// TIA Portal project "Advanced Sorting by height (Working code)" (V17)

(* hardware
DEVICE "S71500/ET200MP-Station_1"  S7-1500 station
   slot 0: "Profilschiene_0"  6ES7 590-1***0-0AA0
   slot 1: "PLC_1"  CPU 1511-1 PN  6ES7 511-1AK00-0AB0  V1.8
   slot 2: "AI 8xU/I/RTD/TC ST_1"  AI 8xU/I/RTD/TC ST  6ES7 531-7KF00-0AB0  V2.0
   slot 3: "AI 8xU/I/RTD/TC ST_2"  AI 8xU/I/RTD/TC ST  6ES7 531-7KF00-0AB0  V2.0
   slot 4: "AI 8xU/I/RTD/TC ST_3"  AI 8xU/I/RTD/TC ST  6ES7 531-7KF00-0AB0  V2.0
   slot 5: "AI 8xU/I/RTD/TC ST_4"  AI 8xU/I/RTD/TC ST  6ES7 531-7KF00-0AB0  V2.0
   slot 6: "DI 16x24VDC BA_1"  DI 16x24VDC BA  6ES7 521-1BH10-0AA0  V1.0
*)

// ===== PLC "PLC_1"  CPU 1511-1 PN =====

VAR_GLOBAL   // PLC tag table "Standard-Variablentabelle"
   "At entry" AT %I0.0 : Bool;
   "Low box" AT %I0.1 : Bool;
   "High box" AT %I0.2 : Bool;
   "At turnable entry" AT %I0.3 : Bool;
   "At load position" AT %I0.4 : Bool;
   "At unload position" AT %I0.5 : Bool;
   "At front" AT %I0.6 : Bool;
   "At right entry" AT %I0.7 : Bool;
   "At left entry" AT %I1.0 : Bool;
   "At right exit" AT %I1.1 : Bool;
   "At left exit" AT %I1.2 : Bool;
   "Start" AT %I1.3 : Bool;
   "Reset" AT %I1.4 : Bool;
   "Stop" AT %I1.5 : Bool;
   "Emergency stop" AT %I1.6 : Bool;
   "Auto" AT %I1.7 : Bool;
   "Feeder Conveyor" AT %Q0.0 : Bool;
   "Entry Conveyor" AT %Q0.1 : Bool;
   "Load" AT %Q0.2 : Bool;
   "Unload" AT %Q0.3 : Bool;
   "Turn" AT %Q0.4 : Bool;
   "Left conveyor" AT %Q0.5 : Bool;
   "Right conveyor" AT %Q0.6 : Bool;
   "Green Indicator" AT %Q0.7 : Bool;
   "Yellow indicator" AT %Q1.0 : Bool;
   "Red indicator" AT %Q1.1 : Bool;
   "Start light" AT %Q1.2 : Bool;
   "Reset light" AT %Q1.3 : Bool;
   "Stop light" AT %Q1.4 : Bool;
   "Counter" AT %Q1.5 : Bool;
   "State 0" AT %M0.0 : Bool;
   "State 1" AT %M0.1 : Bool;
   "State 2" AT %M0.2 : Bool;
   "State 3" AT %M0.3 : Bool;
   "State 4" AT %M0.4 : Bool;
   "Factory IO Running" AT %I2.0 : Bool;
   "State 5" AT %M0.5 : Bool;
   "State 6" AT %M0.6 : Bool;
   "State 10" AT %M0.7 : Bool;
   "Low box detected" AT %M1.0 : Bool;
   "High box detected" AT %M1.1 : Bool;
   "Large box detected" AT %M1.2 : Bool;
   "Tag_1" AT %M2.0 : Bool;
   "Tag_2" AT %M2.1 : Bool;
   "Tag_3" AT %M2.2 : Bool;
   "Tag_6" AT %M2.3 : Bool;
   "Tag_9" AT %M2.4 : Bool;
   "Tag_10" AT %M2.5 : Bool;
   "Tag_11" AT %M2.6 : Bool;
   "Tag_12" AT %M2.7 : Bool;
   "Tag_14" AT %M3.0 : Bool;
   "Tag_15" AT %M3.1 : Bool;
   "Tag_16" AT %M3.2 : Bool;
   "Tag_17" AT %M3.3 : Bool;
   "Tag_18" AT %M3.4 : Bool;
   "Tag_19" AT %M4.0 : Bool;
   "Tag_20" AT %M5.0 : Bool;
END_VAR

FUNCTION "Start/Stop" : Void   // FC1, LAD
{ S7_Optimized_Access := 'TRUE' }
VERSION : 0.1
BEGIN

REGION Network 1: Start System
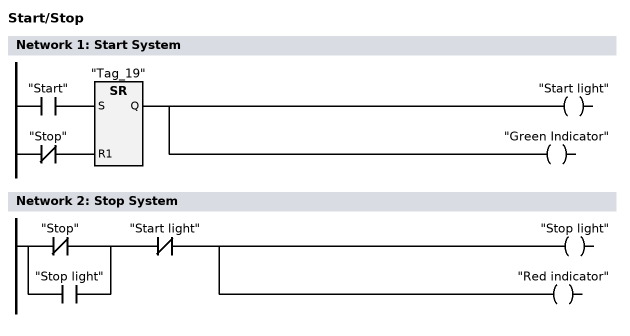
   RUNG wire#powerrail
      Contact( "Start" )
      S_SR(operand := "Tag_19", r1 := wire#w1)
      wire#w2
      Coil( "Start light" )
   END_RUNG
   RUNG wire#powerrail
      I_Contact( "Stop" )
   END_RUNG wire#w1
   RUNG wire#w2
      Coil( "Green Indicator" )
   END_RUNG
   // the same network as SCL:
   IF "Start" THEN
       "Tag_19" := TRUE;   // SR flip-flop
   END_IF;
   IF NOT "Stop" THEN "Tag_19" := FALSE; END_IF;
   "Start light" := "Tag_19";
   "Green Indicator" := "Tag_19";
END_REGION

REGION Network 2: Stop System
   RUNG wire#powerrail
      I_Contact( "Stop" )
      wire#w1
      I_Contact( "Start light" )
      wire#w2
      Coil( "Stop light" )
   END_RUNG
   RUNG wire#powerrail
      Contact( "Stop light" )
   END_RUNG wire#w1
   RUNG wire#w2
      Coil( "Red indicator" )
   END_RUNG
   // the same network as SCL:
   "Stop light" := (NOT "Stop" OR "Stop light") AND NOT "Start light";
   "Red indicator" := "Stop light";
END_REGION
END_FUNCTION

FUNCTION "States" : Void   // FC2, LAD
TITLE = States of the
{ S7_Optimized_Access := 'TRUE' }
VERSION : 0.1
// In this Programm, we will make every actuator is a state, and we will focus on Set Reset conditions, 
// POV : we will not consider which first and which after because it isn't recurrent
   VAR_TEMP   // added for the SCL form of the ladder/FBD networks
      _w1 : Bool;
      _w2 : Bool;
   END_VAR
BEGIN

REGION Network 1: Reset Loop
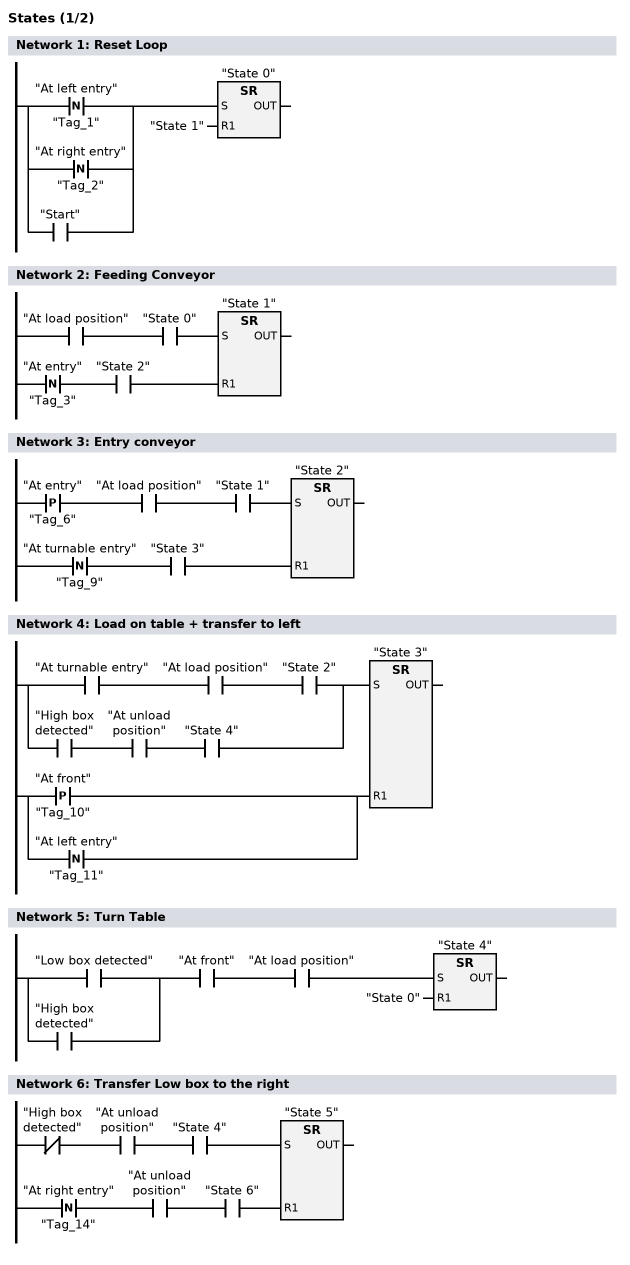
   RUNG wire#powerrail
      N_Contact(operand := "At left entry", bit := "Tag_1")
      wire#w1
      S_SR(operand := "State 0", r1 := "State 1")
   END_RUNG
   RUNG wire#powerrail
      N_Contact(operand := "At right entry", bit := "Tag_2")
   END_RUNG wire#w1
   RUNG wire#powerrail
      Contact( "Start" )
   END_RUNG wire#w1
   // the same network as SCL:
   #_w1 := NOT "At left entry" AND "Tag_1";   // falling edge of "At left entry"
   "Tag_1" := "At left entry";
   #_w2 := NOT "At right entry" AND "Tag_2";   // falling edge of "At right entry"
   "Tag_2" := "At right entry";
   IF #_w1 OR #_w2 OR "Start" THEN
       "State 0" := TRUE;   // SR flip-flop
   END_IF;
   IF "State 1" THEN "State 0" := FALSE; END_IF;
END_REGION

REGION Network 2: Feeding Conveyor
   RUNG wire#powerrail
      Contact( "At load position" )
      Contact( "State 0" )
      S_SR(operand := "State 1", r1 := wire#w1)
   END_RUNG
   RUNG wire#powerrail
      N_Contact(operand := "At entry", bit := "Tag_3")
      Contact( "State 2" )
   END_RUNG wire#w1
   // the same network as SCL:
   #_w1 := NOT "At entry" AND "Tag_3";   // falling edge of "At entry"
   "Tag_3" := "At entry";
   IF "At load position" AND "State 0" THEN
       "State 1" := TRUE;   // SR flip-flop
   END_IF;
   IF #_w1 AND "State 2" THEN "State 1" := FALSE; END_IF;
END_REGION

REGION Network 3: Entry conveyor
   RUNG wire#powerrail
      P_Contact(operand := "At entry", bit := "Tag_6")
      Contact( "At load position" )
      Contact( "State 1" )
      S_SR(operand := "State 2", r1 := wire#w1)
   END_RUNG
   RUNG wire#powerrail
      N_Contact(operand := "At turnable entry", bit := "Tag_9")
      Contact( "State 3" )
   END_RUNG wire#w1
   // the same network as SCL:
   #_w1 := "At entry" AND NOT "Tag_6";   // rising edge of "At entry"
   "Tag_6" := "At entry";
   #_w2 := NOT "At turnable entry" AND "Tag_9";   // falling edge of "At turnable entry"
   "Tag_9" := "At turnable entry";
   IF #_w1 AND "At load position" AND "State 1" THEN
       "State 2" := TRUE;   // SR flip-flop
   END_IF;
   IF #_w2 AND "State 3" THEN "State 2" := FALSE; END_IF;
END_REGION

REGION Network 4: Load on table + transfer to left
   RUNG wire#powerrail
      Contact( "At turnable entry" )
      Contact( "At load position" )
      Contact( "State 2" )
      wire#w1
      S_SR(operand := "State 3", r1 := wire#w2)
   END_RUNG
   RUNG wire#powerrail
      Contact( "High box detected" )
      Contact( "At unload position" )
      Contact( "State 4" )
   END_RUNG wire#w1
   RUNG wire#powerrail
      P_Contact(operand := "At front", bit := "Tag_10")
   END_RUNG wire#w2
   RUNG wire#powerrail
      N_Contact(operand := "At left entry", bit := "Tag_11")
   END_RUNG wire#w2
   // the same network as SCL:
   #_w1 := "At front" AND NOT "Tag_10";   // rising edge of "At front"
   "Tag_10" := "At front";
   #_w2 := NOT "At left entry" AND "Tag_11";   // falling edge of "At left entry"
   "Tag_11" := "At left entry";
   IF ("At turnable entry" AND "At load position" AND "State 2") OR ("High box detected" AND "At unload position" AND "State 4") THEN
       "State 3" := TRUE;   // SR flip-flop
   END_IF;
   IF #_w1 OR #_w2 THEN "State 3" := FALSE; END_IF;
END_REGION

REGION Network 5: Turn Table
   RUNG wire#powerrail
      Contact( "Low box detected" )
      wire#w1
      Contact( "At front" )
      Contact( "At load position" )
      S_SR(operand := "State 4", r1 := "State 0")
   END_RUNG
   RUNG wire#powerrail
      Contact( "High box detected" )
   END_RUNG wire#w1
   // the same network as SCL:
   IF ("Low box detected" OR "High box detected") AND "At front" AND "At load position" THEN
       "State 4" := TRUE;   // SR flip-flop
   END_IF;
   IF "State 0" THEN "State 4" := FALSE; END_IF;
END_REGION

REGION Network 6: Transfer Low box to the right
   RUNG wire#powerrail
      I_Contact( "High box detected" )
      Contact( "At unload position" )
      Contact( "State 4" )
      S_SR(operand := "State 5", r1 := wire#w1)
   END_RUNG
   RUNG wire#powerrail
      N_Contact(operand := "At right entry", bit := "Tag_14")
      Contact( "At unload position" )
      Contact( "State 6" )
   END_RUNG wire#w1
   // the same network as SCL:
   #_w1 := NOT "At right entry" AND "Tag_14";   // falling edge of "At right entry"
   "Tag_14" := "At right entry";
   IF NOT "High box detected" AND "At unload position" AND "State 4" THEN
       "State 5" := TRUE;   // SR flip-flop
   END_IF;
   IF #_w1 AND "At unload position" AND "State 6" THEN "State 5" := FALSE; END_IF;
END_REGION

REGION Network 7: Right conveyor
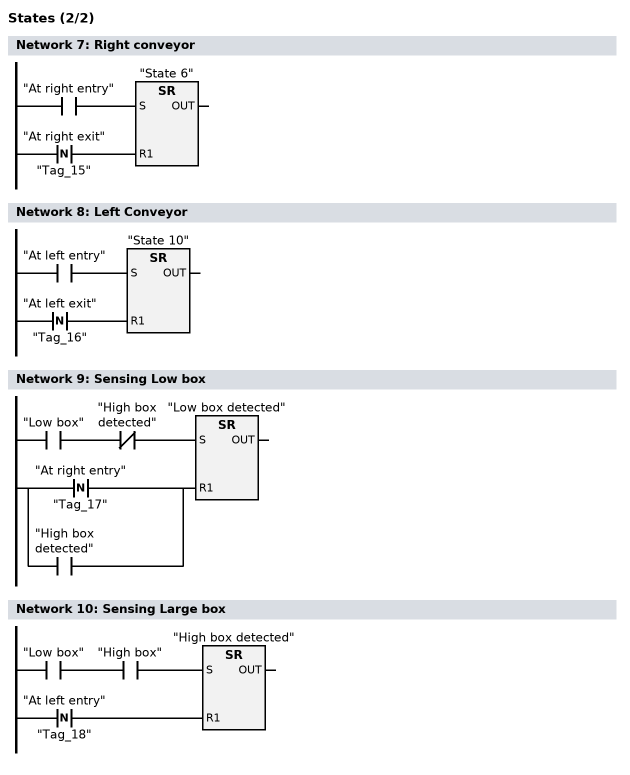
   RUNG wire#powerrail
      Contact( "At right entry" )
      S_SR(operand := "State 6", r1 := wire#w1)
   END_RUNG
   RUNG wire#powerrail
      N_Contact(operand := "At right exit", bit := "Tag_15")
   END_RUNG wire#w1
   // the same network as SCL:
   #_w1 := NOT "At right exit" AND "Tag_15";   // falling edge of "At right exit"
   "Tag_15" := "At right exit";
   IF "At right entry" THEN
       "State 6" := TRUE;   // SR flip-flop
   END_IF;
   IF #_w1 THEN "State 6" := FALSE; END_IF;
END_REGION

REGION Network 8: Left Conveyor
   RUNG wire#powerrail
      Contact( "At left entry" )
      S_SR(operand := "State 10", r1 := wire#w1)
   END_RUNG
   RUNG wire#powerrail
      N_Contact(operand := "At left exit", bit := "Tag_16")
   END_RUNG wire#w1
   // the same network as SCL:
   #_w1 := NOT "At left exit" AND "Tag_16";   // falling edge of "At left exit"
   "Tag_16" := "At left exit";
   IF "At left entry" THEN
       "State 10" := TRUE;   // SR flip-flop
   END_IF;
   IF #_w1 THEN "State 10" := FALSE; END_IF;
END_REGION

REGION Network 9: Sensing Low box
   RUNG wire#powerrail
      Contact( "Low box" )
      I_Contact( "High box detected" )
      S_SR(operand := "Low box detected", r1 := wire#w1)
   END_RUNG
   RUNG wire#powerrail
      N_Contact(operand := "At right entry", bit := "Tag_17")
   END_RUNG wire#w1
   RUNG wire#powerrail
      Contact( "High box detected" )
   END_RUNG wire#w1
   // the same network as SCL:
   #_w1 := NOT "At right entry" AND "Tag_17";   // falling edge of "At right entry"
   "Tag_17" := "At right entry";
   IF "Low box" AND NOT "High box detected" THEN
       "Low box detected" := TRUE;   // SR flip-flop
   END_IF;
   IF #_w1 OR "High box detected" THEN "Low box detected" := FALSE; END_IF;
END_REGION

REGION Network 10: Sensing Large box
   RUNG wire#powerrail
      Contact( "Low box" )
      Contact( "High box" )
      S_SR(operand := "High box detected", r1 := wire#w1)
   END_RUNG
   RUNG wire#powerrail
      N_Contact(operand := "At left entry", bit := "Tag_18")
   END_RUNG wire#w1
   // the same network as SCL:
   #_w1 := NOT "At left entry" AND "Tag_18";   // falling edge of "At left entry"
   "Tag_18" := "At left entry";
   IF "Low box" AND "High box" THEN
       "High box detected" := TRUE;   // SR flip-flop
   END_IF;
   IF #_w1 THEN "High box detected" := FALSE; END_IF;
END_REGION
END_FUNCTION

FUNCTION "Actuators" : Void   // FC3, LAD
{ S7_Optimized_Access := 'TRUE' }
VERSION : 0.1
BEGIN

REGION Network 1: State 0
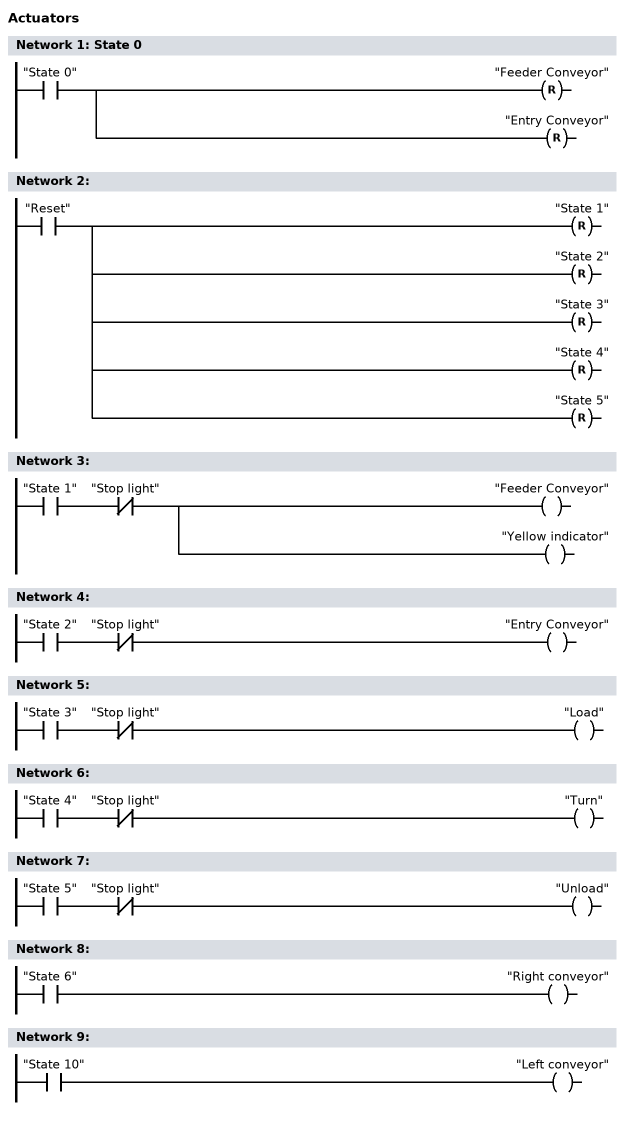
   RUNG wire#powerrail
      Contact( "State 0" )
      wire#w1
      R_Coil( "Feeder Conveyor" )
   END_RUNG
   RUNG wire#w1
      R_Coil( "Entry Conveyor" )
   END_RUNG
   // the same network as SCL:
   IF "State 0" THEN
       "Feeder Conveyor" := FALSE;
       "Entry Conveyor" := FALSE;
   END_IF;
END_REGION

REGION Network 2
   RUNG wire#powerrail
      Contact( "Reset" )
      wire#w1
      R_Coil( "State 1" )
   END_RUNG
   RUNG wire#w1
      R_Coil( "State 2" )
   END_RUNG
   RUNG wire#w1
      R_Coil( "State 3" )
   END_RUNG
   RUNG wire#w1
      R_Coil( "State 4" )
   END_RUNG
   RUNG wire#w1
      R_Coil( "State 5" )
   END_RUNG
   // the same network as SCL:
   IF "Reset" THEN
       "State 1" := FALSE;
       "State 2" := FALSE;
       "State 3" := FALSE;
       "State 4" := FALSE;
       "State 5" := FALSE;
   END_IF;
END_REGION

REGION Network 3
   RUNG wire#powerrail
      Contact( "State 1" )
      I_Contact( "Stop light" )
      wire#w1
      Coil( "Feeder Conveyor" )
   END_RUNG
   RUNG wire#w1
      Coil( "Yellow indicator" )
   END_RUNG
   // the same network as SCL:
   "Feeder Conveyor" := "State 1" AND NOT "Stop light";
   "Yellow indicator" := "Feeder Conveyor";
END_REGION

REGION Network 4
   RUNG wire#powerrail
      Contact( "State 2" )
      I_Contact( "Stop light" )
      Coil( "Entry Conveyor" )
   END_RUNG
   // the same network as SCL:
   "Entry Conveyor" := "State 2" AND NOT "Stop light";
END_REGION

REGION Network 5
   RUNG wire#powerrail
      Contact( "State 3" )
      I_Contact( "Stop light" )
      Coil( "Load" )
   END_RUNG
   // the same network as SCL:
   "Load" := "State 3" AND NOT "Stop light";
END_REGION

REGION Network 6
   RUNG wire#powerrail
      Contact( "State 4" )
      I_Contact( "Stop light" )
      Coil( "Turn" )
   END_RUNG
   // the same network as SCL:
   "Turn" := "State 4" AND NOT "Stop light";
END_REGION

REGION Network 7
   RUNG wire#powerrail
      Contact( "State 5" )
      I_Contact( "Stop light" )
      Coil( "Unload" )
   END_RUNG
   // the same network as SCL:
   "Unload" := "State 5" AND NOT "Stop light";
END_REGION

REGION Network 8
   RUNG wire#powerrail
      Contact( "State 6" )
      Coil( "Right conveyor" )
   END_RUNG
   // the same network as SCL:
   "Right conveyor" := "State 6";
END_REGION

REGION Network 9
   RUNG wire#powerrail
      Contact( "State 10" )
      Coil( "Left conveyor" )
   END_RUNG
   // the same network as SCL:
   "Left conveyor" := "State 10";
END_REGION
END_FUNCTION

FUNCTION "MHJ-PLC-Lab-Function-S71500" : Void   // FC9000, SCL
{ S7_Optimized_Access := 'TRUE' }
VERSION : 0.1
   VAR_TEMP
      Value : Byte;
      ForCounter : Int;
   END_VAR
   VAR CONSTANT
      Value_01_DW : DWord := 16#1223_5486;
      Value_02_DW : DWord := 16#A6C9_D1F5;
   END_VAR
BEGIN

   #Value:=PEEK(area := 16#82,
        dbNumber := 0,
        byteOffset := 511);
   #Value := #Value + 1;

   POKE(area := 16#82,
        dbNumber := 0,
        byteOffset := 511,
        value := #Value);

   POKE(area := 16#82,
        dbNumber := 0,
        byteOffset := 1016,
        value := #Value_01_DW);
   POKE(area := 16#82,
        dbNumber := 0,
        byteOffset := 1020,
        value := #Value_02_DW);

   FOR #ForCounter := 0 TO 63 DO
       #Value:=PEEK(area := 16#1,
            dbNumber := 0,
            byteOffset := #ForCounter);
       POKE(area := 16#81,
            dbNumber := 0,
            byteOffset := #ForCounter,
            value := #Value);
   END_FOR;
   #Value := PEEK(area := 16#1,
                  dbNumber := 0,
                  byteOffset := 512);
   POKE(area := 16#82,
        dbNumber := 0,
        byteOffset := 512,
        value := #Value);
END_FUNCTION

ORGANIZATION_BLOCK "Main"   // OB1, LAD, ProgramCycle
TITLE = "Main Program Sweep (Cycle)"
{ S7_Optimized_Access := 'TRUE' }
VERSION : 0.1
   VAR_INPUT
      Initial_Call : Bool;   // Initial call of this OB
      Remanence : Bool;   // =True, if remanent data are available
   END_VAR
BEGIN

REGION Network 1: This network is for connecting TIA V-16 with Factory I/O, do not delete.
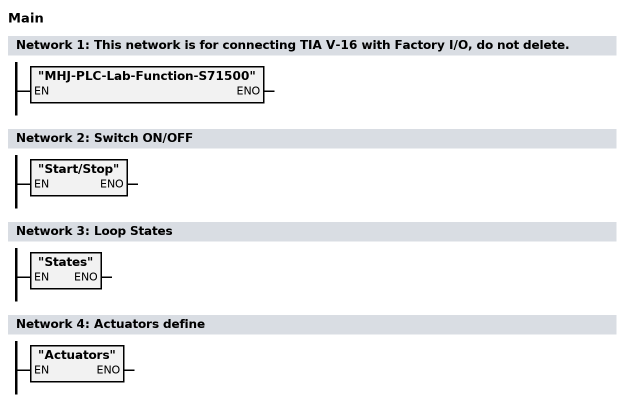
   RUNG wire#powerrail
      "MHJ-PLC-Lab-Function-S71500"()
   END_RUNG
   // the same network as SCL:
   "MHJ-PLC-Lab-Function-S71500"();
END_REGION

REGION Network 2: Switch ON/OFF
   RUNG wire#powerrail
      "Start/Stop"()
   END_RUNG
   // the same network as SCL:
   "Start/Stop"();
END_REGION

REGION Network 3: Loop States
   RUNG wire#powerrail
      "States"()
   END_RUNG
   // the same network as SCL:
   "States"();
END_REGION

REGION Network 4: Actuators define
   RUNG wire#powerrail
      "Actuators"()
   END_RUNG
   // the same network as SCL:
   "Actuators"();
END_REGION
END_ORGANIZATION_BLOCK

ORGANIZATION_BLOCK "Startup"   // OB100, LAD, Startup
TITLE = "Complete Restart"
{ S7_Optimized_Access := 'TRUE' }
VERSION : 0.1
   VAR_INPUT
      LostRetentive : Bool;   // True if retentive data are lost
      LostRTC : Bool;   // True if date and time are lost
   END_VAR
   VAR_TEMP   // added for the SCL form of the ladder/FBD networks
      _w1 : Bool;
      _w2 : Bool;
   END_VAR
BEGIN

REGION Network 1
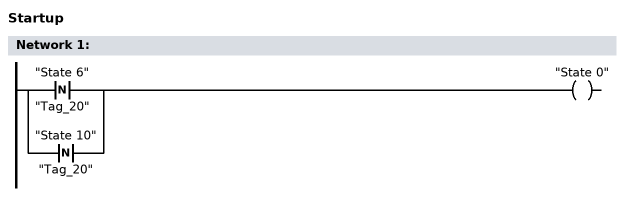
   RUNG wire#powerrail
      N_Contact(operand := "State 6", bit := "Tag_20")
      wire#w1
      Coil( "State 0" )
   END_RUNG
   RUNG wire#powerrail
      N_Contact(operand := "State 10", bit := "Tag_20")
   END_RUNG wire#w1
   // the same network as SCL:
   #_w1 := NOT "State 6" AND "Tag_20";   // falling edge of "State 6"
   "Tag_20" := "State 6";
   #_w2 := NOT "State 10" AND "Tag_20";   // falling edge of "State 10"
   "Tag_20" := "State 10";
   "State 0" := #_w1 OR #_w2;
END_REGION
END_ORGANIZATION_BLOCK